*)
IF X > 20.0 THEN
	SIGMOID := 1.0;
ELSIF x < -85.0 THEN
	SIGMOID := 0.0;
ELSE
	SIGMOID := 1.0 / (1.0 + EXP(-X));
END_IF;


(* revision history
hm	10.12.2007		rev 1.0
	original version

hm	11. mar. 2008		rev 1.1
	extended range of valid inputs to +inv / -inv

hm 10. mar. 2009		rev 1.2
	real constants updated to new systax using dot																																																																																																																																																																																																																																																																																																																																																																																																																																																																																																																																																																																																																																																																																																																																																																																																																																																																																																																																																																																																																																																											

*)
END_FUNCTION

(* POU Mathematical/SIGN_I, ST *)
FUNCTION SIGN_I : BOOL
VAR_INPUT
	IN : DINT;
END_VAR


(*
version 1.3	27. oct. 2008
programmer 	hugo
tested by	tobias

this function return true if the integer input is negative

*)
SIGN_I := in.31;

(* revision history
hm 3.3.2007	rev 1.1
	changed method of function for better compatibility to other systems

hm	1.12.2007	rev 1.2
	changed code to improve performance

hm	27. oct. 2008	rev 1.3
	changed type of input to dint

*)
END_FUNCTION

(* POU Engineering/automation/SIGNAL, ST *)
FUNCTION_BLOCK SIGNAL
VAR_INPUT
	IN : BOOL;
	SIG : BYTE;
	TS : TIME;
END_VAR
VAR_OUTPUT
	Q : BOOL;
END_VAR
VAR
	tx: DWORD;
	step: BYTE;
END_VAR
VAR CONSTANT
	one : BYTE := 1;
END_VAR

(*
version 1.0	13 dec 2007
programmer 	hugo
tested by		tobias

this function generates an output signal according to a bit pattern SIG.
the patter is shifted to the output in time steps of TS.
ts defaults to 128 ms if not specified.
*)
IF in THEN
	(* an alarm is present read system time first *)
	tx := T_PLC_MS();
	(* calculate the step counter which is the lowest 3 bits of (time / ts) *)
	IF ts > t#0s THEN
		step := DWORD_TO_BYTE(tx / TIME_TO_DWORD(ts) AND 16#0000_0007);
	ELSE
		step := DWORD_TO_BYTE(SHR(tx,7) AND 16#0000_0007);
	END_IF;
	(* convert the value 0-7 in step into one bit only (bit 0-7) *)
	step := SHL(one,step);
	(* generate the output signal *)
	Q := (step AND sig) > 0;
ELSE
	Q := FALSE;
END_IF;

(* revision history
hm	13.12.2007		rev 1.0
	original version

*)
END_FUNCTION_BLOCK

(* POU Engineering/automation/SIGNAL_4, ST *)
FUNCTION_BLOCK SIGNAL_4
VAR_INPUT
	IN1 : BOOL;
	IN2 : BOOL;
	IN3 : BOOL;
	IN4 : BOOL;
	TS : TIME;
END_VAR
VAR_INPUT CONSTANT
	S1 : BYTE := 2#1111_1111;
	S2 : BYTE := 2#1111_0000;
	S3 : BYTE := 2#1010_1010;
	S4 : BYTE := 2#1010_0000;
END_VAR
VAR_OUTPUT
	Q : BOOL;
END_VAR
VAR
	sig : SIGNAL;
END_VAR

(*
version 1.0	13 dec 2007
programmer 	hugo
tested by		tobias

this function generates one out of 4 signals specified by bit patterns S1 .. S4.
the selected pattern will be shifted with the step time TS.
In1 has higher priority then In2 which has higher priority then IN3 and in4 has the lowest priority.
ts defaults to 128 ms if not specified.
*)
(* an alarm is present read system time first *)
(* check if an alarm is present if yes set sig to the alarm pattern otherwise exit the routine *)
IF in1 THEN
	sig(in := TRUE, sig := s1, TS := TS);
ELSIF in2 THEN
	sig(in := TRUE, sig := s2, TS := TS);
ELSIF in3 THEN
	sig(in := TRUE, sig := s3, TS := TS);
ELSIF in4 THEN
	sig(in := TRUE, sig := s4, TS := TS);
ELSE
	sig(in := FALSE);
END_IF;

(* set the output *)
Q := sig.Q;


(* revision history
hm	13.12.2007		rev 1.0
	original version

*)
END_FUNCTION_BLOCK

(* POU Mathematical/SINC, ST *)
FUNCTION SINC : REAL
VAR_INPUT
	X : REAL;
END_VAR


(*
version 1.2	10. mar. 2009
programmer 	hugo
tested by		tobias

this function calculates the sinc function.

*)
IF X = 0.0 THEN
	SINC := 1.0;
ELSE
	SINC := SIN(x) / x;
END_IF;


(* revision histroy
hm	11. mar. 2008	rev 1.0
	original version

hm	1.12.2007	rev 1.1
	changed code to improove performance

hm 10. mar. 2009	rev 1.2
	real constants updated to new systax using dot																																																																																																																																																																																																																																																																																																																																																																																																																																																																																																																																																																																																																																																																																																																																																																																																																																																																																																																																																																																																																																																											

*)
END_FUNCTION

(* POU Mathematical/Geometry/SPHERE_V, ST *)
FUNCTION SPHERE_V : REAL
VAR_INPUT
	rx : REAL;
END_VAR


(*
version 1.2	22. feb 2008
programmer 	hugo
tested by		tobias

sphere_V calculates the Volume of a Sphere


*)
sphere_V := 4.188790205 * Rx * RX * RX;

(* revision histroy
hm	16. oct 2007	rev 1.0
	original version

hm	4. dec 2007		rev 1.1
	changed code for better performance

hm	22. feb 2008		rev 1.2
	changed code for better performance
*)
END_FUNCTION

(* POU Logic/memory/STACK_16, ST *)
FUNCTION_BLOCK STACK_16
VAR_INPUT
	Din : DWORD;
	E : BOOL := TRUE;
	RD : BOOL;
	WD : BOOL;
	RST : BOOL;
END_VAR
VAR_OUTPUT
	Dout : DWORD;
	EMPTY : BOOL := TRUE;
	FULL : BOOL;
END_VAR
VAR
	stack : ARRAY[0..n] OF DWORD;
	pt : INT;
END_VAR
VAR CONSTANT
	n : INT := 15;	(* changing this value will chage the number of stored elements in the fifo *)
END_VAR


(*
version 2.0	25. jul 2009
programmer 	hugo
tested by		oscat

16 Dword STACK memory

*)
IF RST THEN
	(* asynchronous reset for the fifo *)
	pt := 0;
	EMPTY := TRUE;
	FULL := FALSE;
	Dout := 0;
ELSIF E THEN
	IF NOT EMPTY AND RD THEN
		(* read one element *)
		pt := pt - 1;
		Dout := stack[pt];
		EMPTY := pt = 0;
		FULL := FALSE;
	END_IF;
	IF NOT FULL AND WD THEN
		(* write one element *)
		stack[pt] := Din;
		pt := pt + 1;
		FULL := pt > n;
		EMPTY := FALSE;
	END_IF;
END_IF;


(* revision history
hm	4. aug. 2006	rev 1.0
	original version

hm	19. feb 2008	rev 1.1
	performance improvements

hm	17. oct. 2008	rev 1.2
	deleted unnecessary init with 0

hm	27. oct. 2008	rev 1.3
	optimized performance

hm	25. jul 2009	rev 2.0
	changed inputs to allow simultsaneous read and write
*)
END_FUNCTION_BLOCK

(* POU Logic/memory/STACK_32, ST *)
FUNCTION_BLOCK STACK_32
VAR_INPUT
	Din : DWORD;
	E : BOOL := TRUE;
	RD : BOOL;
	WD : BOOL;
	RST : BOOL;
END_VAR
VAR_OUTPUT
	Dout : DWORD;
	EMPTY : BOOL := TRUE;
	FULL : BOOL;
END_VAR
VAR
	stack : ARRAY[0..n] OF DWORD;
	pt : INT;
END_VAR
VAR CONSTANT
	n : INT := 31;	(* changing this value will chage the number of stored elements in the fifo *)
END_VAR


(*
version 2.0	25. jul 2009
programmer 	hugo
tested by		oscat

32 Dword STACK memory
*)
IF RST THEN
	(* asynchronous reset for the fifo *)
	pt := 0;
	EMPTY := TRUE;
	FULL := FALSE;
	Dout := 0;
ELSIF E THEN
	IF NOT EMPTY AND RD THEN
		(* read one element *)
		pt := pt - 1;
		Dout := stack[pt];
		EMPTY := pt = 0;
		FULL := FALSE;
	END_IF;
	IF NOT FULL AND WD THEN
		(* write one element *)
		stack[pt] := Din;
		pt := pt + 1;
		FULL := pt > n;
		EMPTY := FALSE;
	END_IF;
END_IF;


(* revision history
hm	4. aug. 2006	rev 1.0
	original version

hm	19. feb 2008	rev 1.1
	performance improvements

hm	17. oct. 2008	rev 1.2
	deleted unnecessary init with 0

ks	27. oct. 2008	rev 1.3
	optimized performance

hm	25. jul 2009	rev 2.0
	changed inputs to allow simultsaneous read and write

*)
END_FUNCTION_BLOCK

(* POU Engineering/signal processing/STAIR, ST *)
FUNCTION STAIR : REAL
VAR_INPUT
	X : REAL;
	D : REAL;
END_VAR


(*
version 1.4	10. mar. 2009
programmer 	oscat
tested by		tobias

the function stair converts an anlog input signal to a staircase like output.
D is the step width for the output signal.
if D = 0 then the output follows the input without a chage.
*) 
IF D > 0.0 THEN
	STAIR := DINT_TO_REAL(REAL_TO_DINT(X / D)) * D;
ELSE
	STAIR := X;
END_IF;



(* revision history
hm	28 jan 2007		rev 1.0
	original version

hm	27 dec 2007		rev 1.1
	changed code for better performance

hm	6. jan 2008		rev 1.2
	further performance improvement

hm	26. oct. 2008		rev 1.3
	optimized code

hm	10. mar. 2009	rev 1.4
	real constants updated to new systax using dot

*)
END_FUNCTION

(* POU Engineering/signal processing/STAIR2, ST *)
FUNCTION_BLOCK STAIR2
VAR_INPUT
	X : REAL;
	D : REAL;
END_VAR
VAR_OUTPUT
	Y: REAL;
END_VAR


(*
version 1.4	10. mar. 2009
programmer 	hugo
tested by		oscat

the function stair2 converts an anlog input signal to a staircase like output.
D is the step width for the output signal. the output will use D as a hysteresis for a stairchange.
if D = 0 then the output follows the input without a chage.
*) 
IF D > 0.0 THEN
	IF X >= Y + D OR X <= Y - D THEN Y := FLOOR(X/D) * D; END_IF;
ELSE
	Y := X;
END_IF;



(* revision history
hm	28 jan 2007		rev 1.0
	original version

hm	27. dec 2007	rev 1.1
	changed code for better performance

hm	30. jun. 2008	rev 1.2
	added type conversions to avoid warnings under codesys 3.0																																																																																																																																																																																																																																																											

ks	26. oct. 2008	rev 1.3
	improved code

hm	10. mar. 2009	rev 1.4
	real constants updated to new systax using dot

*)
END_FUNCTION_BLOCK

(* POU Logic/FF pulse triggered/STORE_8, ST *)
FUNCTION_BLOCK STORE_8
VAR_INPUT
	Set : BOOL;
	D0,D1, D2, D3, D4, D5, D6, D7 : BOOL;
	Clr : BOOL;
	Rst : BOOL;
END_VAR
VAR_OUTPUT
	Q0, Q1, Q2, Q3, Q4, Q5, Q6, Q7 : BOOL;
END_VAR
VAR
	edge: BOOL;
END_VAR

(*
version 1.2	14. mar. 2009
programmer 	hugo
tested by		oscat

Store_4 stores up to 4 boolean inputs until a reset is clearing the outputs.
the respective output is set with a true at the respective input and stays true until a reset is generated.
a set input is used to set all outputs true at the same time, independent of their inputs.
a clear input is used to reset only the lowest priority of the outputs one at a time.
the lowest priority is q3.

*)
IF rst OR set THEN
	q0 := NOT rst;
	q1 := q0;
	q2 := q0;
	q3 := q0;
	q4 := q0;
	q5 := q0;
	q6 := q0;
	q7 := q0;
ELSE
	IF D0 THEN Q0 := TRUE; END_IF;
	IF D1 THEN Q1 := TRUE; END_IF;
	IF D2 THEN Q2 := TRUE; END_IF;
	IF D3 THEN Q3 := TRUE; END_IF;
	IF D4 THEN Q4 := TRUE; END_IF;
	IF D5 THEN Q5 := TRUE; END_IF;
	IF D6 THEN Q6 := TRUE; END_IF;
	IF D7 THEN Q7 := TRUE; END_IF;

	IF clr AND NOT edge THEN
		IF q0 THEN q0 := FALSE;
		ELSIF q1 THEN q1 := FALSE;
		ELSIF q2 THEN q2 := FALSE;
		ELSIF q3 THEN q3 := FALSE;
		ELSIF q4 THEN q4 := FALSE;
		ELSIF q5 THEN q5 := FALSE;
		ELSIF q6 THEN q6 := FALSE;
		ELSE q7 := FALSE;
		END_IF;
	END_IF;
	edge := clr;
END_IF;


(* revision history
hm	25.12.2007	rev 1.0
	original version

hm	30. oct. 2008	rev 1.1
	optimized performance

hm	14. mar. 2009	rev 1.2
	removed double assignments

*)
END_FUNCTION_BLOCK

(* POU Logic/gate logic/SWAP_BYTE, ST *)
FUNCTION SWAP_BYTE : WORD
VAR_INPUT
	IN : WORD;
END_VAR


(*
version 1.0	4 feb 2008
programmer 	hugo
tested by		tobias

This function swaps the high and low byte of the word in.

*)
SWAP_BYTE := ROL(in,8);


(* revision history
hm		4. feb 2008	rev 1.0
	original version

*)
END_FUNCTION

(* POU Logic/gate logic/SWAP_BYTE2, ST *)
FUNCTION SWAP_BYTE2 : DWORD
VAR_INPUT
	IN : DWORD;
END_VAR


(*
version 1.0	4 feb 2008
programmer 	hugo
tested by		tobias

This function reverses the byte order in the dword.

*)
Swap_Byte2 := (ROR(in,8) AND 16#FF00FF00) OR (ROL(in,8) AND 16#00FF00FF);

(* revision history
hm		4. feb 2008	rev 1.0
	original version

*)
END_FUNCTION

(* POU Mathematical/TANC, ST *)
FUNCTION TANC : REAL
VAR_INPUT
	X : REAL;
END_VAR


(*
version 1.1	10. mar. 2009
programmer 	hugo
tested by		oscat

this function calculates the tanc function.

*)
IF X = 0.0 THEN
	TANC := 1.0;
ELSE
	TANC := TAN(x) / x;
END_IF;


(* revision histroy
hm	23. oct. 2008	rev 1.0
	original version

hm 10. mar. 2009	rev 1.1
	real constants updated to new systax using dot																																																																																																																																																																																																																																																																																																																																																																																																																																																																																																																																																																																																																																																																																																																																																																																																																																																																																																																																																																																																																																																											

*)
END_FUNCTION

(* POU Mathematical/TANH, ST *)
FUNCTION TANH : REAL
VAR_INPUT
	X : REAL;
END_VAR


(*
version 1.3	10. mar. 2009
programmer 	hugo
tested by		tobias

this function calculates the tangens hyperbolicus

*)
IF X > 20.0 THEN
	TANH := 1.0;
ELSIF X < -20.0 THEN
	TANH := -1.0;
ELSE
	TANH := 1.0 - 2.0 / (EXP(2.0 * x) + 1.0);
END_IF;


(* revision hisdtory
hm		12.1.2007		rev 1.0
	original version

hm		1.12.2007		rev 1.1
	changed code to improve performance

hm		10. mar 2008	rev 1.2
	corrected an error in formula
	extended range of valid inputs to +/- INV

hm 10. mar. 2009	rev 1.3
	real constants updated to new systax using dot																																																																																																																																																																																																																																																																																																																																																																																																																																																																																																																																																																																																																																																																																																																																																																																																																																																																																																																																																																																																																																																											

*)
END_FUNCTION

(* POU Engineering/measurements/TC_MS, ST *)
FUNCTION_BLOCK TC_MS

VAR_OUTPUT
	TC : DWORD;
END_VAR
VAR
	init: BOOL;
	tx: DWORD;
	last: DWORD;
END_VAR

(*
	version 1.0	13 mar 2008
	programmer 	hugo
	tested by		tobias

TC_MS delivers the time it was last called on the output TC in Milliseconds.

*)
(* read system timer *)
tx := T_PLC_MS();

IF NOT init THEN
	init := TRUE;
	TC := 0;
ELSE
	tc := tx - last;
END_IF;
last := tx;

(* revision history
hm		13. mar. 2008	rev 1.0
	original version

*)
END_FUNCTION_BLOCK

(* POU Engineering/measurements/TC_US, ST *)
FUNCTION_BLOCK TC_US

VAR_OUTPUT
	TC : DWORD;
END_VAR
VAR
	init: BOOL;
	tx: DWORD;
	last: DWORD;
END_VAR

(*
	version 1.0	13 mar 2008
	programmer 	hugo
	tested by		tobias

TC_US delivers the time it was last called on the output TC in Microseconds.

*)
(* read system timer *)
tx := T_PLC_US();

IF NOT init THEN
	init := TRUE;
	TC := 0;
ELSE
	tc := tx - last;
END_IF;
last := tx;

(* revision history
hm		13. mar. 2008	rev 1.0
	original version

*)
END_FUNCTION_BLOCK

(* POU Engineering/sensor/TEMP_NI, ST *)
FUNCTION TEMP_NI : REAL
VAR_INPUT
	Res : REAL;
	R0 : REAL;
END_VAR


(*
version 1.5	10. mar. 2009
programmer 	hugo
tested by		tobias

this function returns the temperature for a nickel sensor in a range from -60..+180 °C *)
TEMP_NI := (SQRT(0.30085225 - 2.66E-3 * (R0 - Res)) - 0.5485) * 751.8796992;


(* revision history

hm 24.1.2007		rev 1.1
	deleted unused variable A, B, C

hm 10.9.2007		rev 1.2
	changed accuracy to 0.02 degrees to improove performace

hm 17. 12 2007	rev 1.3
	improovements for better performance and higher accuracy

hm	6. jan 2008	rev 1.4
	further performance improvement

hm	10. mar. 2009	rev 1.5
	removed nested comments

*)
END_FUNCTION

(* POU Engineering/sensor/TEMP_NTC, ST *)
FUNCTION TEMP_NTC : REAL
VAR_INPUT
	RES : REAL;
	RN : REAL;
	B : REAL;
END_VAR


(*
version 1.1	11. mar. 2009
programmer 	hugo
tested by		tobias

this function returs the temperature for a NTC sensor for a range from 0..85 °C.
RN is the resistance at 25 °C and B is a constant for the given sensor.

*)
IF res > 0.0 THEN
	TEMP_NTC := B * 298.15 / (B + LN(RES / RN) * 298.15) -273.15;
END_IF;


(* revision history

hm 30. dec. 2008	rev 1.0
	original version

hm	11. mar. 2009	rev 1.1
	changed real constants to use dot syntax

*)
END_FUNCTION

(* POU Engineering/sensor/TEMP_PT, ST *)
FUNCTION TEMP_PT : REAL
VAR_INPUT
	Res : REAL;
	R0 : REAL;
END_VAR
VAR CONSTANT
	A : REAL := 3.9083E-3 ;
	B : REAL := -5.775E-7;
	accuracy : REAL := 0.01;
END_VAR
VAR
	step: REAL := 50.0;
	X: REAL;
	Y: REAL;
	t1: REAL;
	pt : POINTER TO DWORD;
END_VAR

(*
version 1.7	11. mar. 2009
programmer 	hugo
tested by		oscat

this function returs the temperature for a platinum sensor for a range from -200..+850 °C *)
X := A * R0;
Y := B * R0;
IF Res >= R0 THEN
	t1 := X * X - 4.0 * Y * (R0 - Res);
	IF t1 < 0.0 THEN
		TEMP_PT := 10000.0;
	ELSE
		TEMP_PT := (-X + SQRT(t1)) / (2.0 * Y);
	END_IF;
ELSE
	pt := ADR(step);
	(* since the formula cannot be solved this is a successive approximation *)
	TEMP_PT := -100.0;
	WHILE step > accuracy DO
		(* test if result greater or less *)
		IF RES_PT(TEMP_PT, R0) < res THEN TEMP_PT := TEMP_PT + step; ELSE TEMP_PT := TEMP_PT - step; END_IF;
		pt^ := pt^ - 8388608;  (* this is a super fast divide by 2 method for non floating point CPUs *)
		(* the alternative code: step := step * 0.5; *)
	END_WHILE;
END_IF;

(* revision history

rev 1.1 hm 24.1.2007	
	deleted unused variable C

rev 1.2 hm 10.9.2007
	reduced accuracy to 0.02 to shorten execution time

rev 1.3	hm	2. dec 2007
	changed code for better performance

rev	1.4	hm	23. dec 2007
	avoid a negative square root if input values are wrong

rev 1.5 hm	5. jan 2008
	replaced / 2 with * 0.5 for better performance

hm	31. oct. 2008	rev 1.6
	improved performance

hm	11. mar. 2009	rev 1.7
	changed real constants to use dot syntax

*)
END_FUNCTION

(* POU Engineering/sensor/TEMP_SI, ST *)
FUNCTION TEMP_SI : REAL
VAR_INPUT
	Res : REAL;
	RS : REAL;
	TS : REAL;
END_VAR


(*
version 1.5	10. mar. 2009
programmer 	hugo
tested by		tobias

this function returs the temperature for a silicon sensor for a range from -60..+180 °C
for example KTY10 RS at TS normally 25 °C
*)
TEMP_SI := (-7.64E-3 + SQRT(Res / RS * 6.64E-5 - 0.803E-5)) * 30120.48193 + TS;



(* revision history

hm 24.1.2007		rev 1.1
	the function would only work for TS = 25, now it works for other values of ts.

hm 10.9.2007		rev 1.2
	changed the function to use successive approcimation to avoid an error generated by a sqrt from a negative result.
	changed accuracy to 0.02 degrees to shorten execution time

hm 17. 12 2007	rev 1.3
	improovements for better performance

hm	6. jan 2008	rev 1.4
	further performance improvement

hm	10. mar. 2009	rev 1.5
	removed nested comments

*)
END_FUNCTION

(* POU Engineering/conversion/TEMPERATURE, ST *)
FUNCTION_BLOCK TEMPERATURE
VAR_INPUT
	K : REAL;
	C : REAL := -273.15;
	F : REAL := -459.67;
	Re : REAL := -218.52;
	Ra : REAL;
END_VAR
VAR_OUTPUT
	YK : REAL;
	YC : REAL;
	YF : REAL;
	YRe : REAL;
	YRa : REAL;
END_VAR


(*
version 1.0	21 feb 2008
programmer 	hugo
tested by	oscat

this function converts different temperature units
any unused input can simply be left open.
different inputs connected at the same time will be added up.

*)
YK := K + (C + 273.15) + (F + 459.67) * 0.555555555555 + (Re * 1.25 + 273.15) + (Ra * 0.555555555555);
YC := YK -273.15;
YF := YK * 1.8 - 459.67;
YRe := (YK - 273.15) * 0.8;
YRa := YK * 1.8;


(* revision history
hm	21. feb. 2008	rev 1.0
	original version

*)
END_FUNCTION_BLOCK

(* POU X_TEST/TEST_ARRAY_SORT, ST *)
FUNCTION_BLOCK TEST_ARRAY_SORT
VAR_INPUT
END_VAR
VAR_OUTPUT
END_VAR
VAR CONSTANT
	array_max : INT := 999;
END_VAR
VAR
	buffer : ARRAY[0..array_max] OF REAL;
	i: INT;
	tx: TIME;
	t_sort : TIME;
END_VAR
(* prefill array *)
buffer[0] := 0.0;
buffer[1] := 1.0;
buffer[2] := 0.0;
buffer[3] := -100.0;
buffer[4] := 100.0;

FOR i := 5 TO ARRAY_MAX DO
	buffer[i] := INT_TO_REAL(i)-20.0;
END_FOR;

_ARRAY_SHUFFLE(ADR(buffer), SIZEOF(buffer));
tx := TIME();
_ARRAY_SORT(ADR(buffer), SIZEOF(buffer));
t_sort := TIME() - tx;
END_FUNCTION_BLOCK

(* POU X_TEST/TEST_CRC_GEN, ST *)
FUNCTION_BLOCK TEST_CRC_GEN
VAR_INPUT
END_VAR
VAR_OUTPUT
	ERROR : BOOL;
	info : STRING (10);
END_VAR
VAR
	BUFFER : ARRAY[0..8] OF BYTE := 16#31, 16#32, 16#33, 16#34, 16#35, 16#36, 16#37, 16#38, 16#39;
	pt : POINTER TO ARRAY[0..100] OF BYTE;
	size : INT;
	erg: DWORD;
END_VAR
pt := ADR(buffer);
size := SIZEOF(buffer);

erg := CRC_GEN(pt, size, 3, 16#3, 16#7, TRUE, TRUE, 16#0);
IF erg <> 16#6 THEN
	error := TRUE;
	info := 'CRC-3/ROHC';
END_IF;

erg := CRC_GEN(pt, size, 5, 16#9, 16#9, FALSE, FALSE, 16#0);
IF erg <> 16#0 THEN
	error := TRUE;
	info := 'CRC-5/EPC';
END_IF;

erg := CRC_GEN(pt, size, 6, 16#19, 16#0, TRUE, FALSE, 16#0);
IF erg <> 16#19 THEN
	error := TRUE;
	info := 'CRC-6/DARC';
END_IF;

erg := CRC_GEN(pt, size, 7, 16#4F, 16#7F, TRUE, TRUE, 16#0);
IF erg <> 16#53 THEN
	error := TRUE;
	info := 'CRC-7/ROHC';
END_IF;

erg := CRC_GEN(pt, size, 8, 16#1D, 16#FD, FALSE, FALSE, 16#0);
IF erg <> 16#7E THEN
	error := TRUE;
	info := 'CRC-8/I-CODE';
END_IF;

erg := CRC_GEN(pt, size, 10, 16#233, 16#000, FALSE, FALSE, 16#0);
IF erg <> 16#199 THEN
	error := TRUE;
	info := 'CRC-10';
END_IF;

erg := CRC_GEN(pt, size, 12, 16#80F, 16#000, FALSE, TRUE, 16#0);
IF erg <> 16#DAF THEN
	error := TRUE;
	info := 'CRC-12/3GPP';
END_IF;

erg := CRC_GEN(pt, size, 14, 16#0805, 16#000, TRUE, TRUE, 16#0);
IF erg <> 16#082D  THEN
	error := TRUE;
	info := 'CRC-14/DARC';
END_IF;

erg := CRC_GEN(pt, size, 15, 16#4599, 16#000, FALSE, FALSE, 16#0);
IF erg <> 16#059E  THEN
	error := TRUE;
	info := 'CRC-15';
END_IF;

erg := CRC_GEN(pt, size, 16, 16#8BB7, 16#000, FALSE, FALSE, 16#0);
IF erg <> 16#D0DB  THEN
	error := TRUE;
	info := 'CRC-16/T10-DIF';
END_IF;

erg := CRC_GEN(pt, size, 24, 16#5D6DCB, 16#ABCDEF, FALSE, FALSE, 16#0);
IF erg <> 16#1F23B8  THEN
	error := TRUE;
	info := 'CRC-24/FLEXRAY-B';
END_IF;

erg := CRC_GEN(pt, size, 32, 16#04C11DB7, 16#FFFFFFFF, TRUE, TRUE, 16#0);
IF erg <> 16#340BC6D9  THEN
	error := TRUE;
	info := 'JAMCRC';
END_IF;



(*
   Name   : "CRC-82/DARC"
   Width  : 82
   Poly   : 0308C0111011401440411
   Init   : 000000000000000000000
   RefIn  : True
   RefOut : True
   XorOut : 000000000000000000000
   Check  : 09EA83F625023801FD612
	pt : POINTER TO ARRAY[1..32000] OF BYTE;
	size : UINT;
	Polynom_L : DWORD;
	Polynom_32 : BOOL;
	init: DWORD;
	XOR_out : DWORD;
	rev_in : BOOL;
	rev_out : BOOL;

*)
END_FUNCTION_BLOCK

(* POU X_TEST/test_date, ST *)
FUNCTION_BLOCK test_date
VAR_INPUT
END_VAR
VAR_OUTPUT
	error: BOOL;
END_VAR
VAR
	test : DWORD;
	c_date : DATE;
	x_date : DATE;
	c_day : INT;
	c_month : INT;
	c_year : INT;
	d_str : STRING;
END_VAR
c_date := DWORD_TO_DATE(test);
d_str := DATE_TO_STRING(c_date);
c_year := STRING_TO_INT(MID(d_str, 4, 3));
c_month := STRING_TO_INT(MID(d_str, 2, 8));
c_day := STRING_TO_INT(MID(d_str, 2, 11));


(* test leap_day *)
IF LEAP_DAY(c_date)  XOR (c_day = 29 AND c_month = 2) THEN error := TRUE; END_IF;

(* test set_date *)
x_date := SET_DATE(c_year, c_month, c_day);
IF x_date <> c_date THEN error := TRUE; END_IF;

(* test year_end *)
IF SET_DATE(c_year, 12, 31) <> YEAR_END(c_year) THEN error := TRUE; END_IF;

(* test year begin  and day_of_year *)
x_date := YEAR_BEGIN(c_year);
IF SET_DATE(c_year, 1, 1) <> x_date THEN error := TRUE; END_IF;
(* test day_of_year *)
IF UDINT_TO_DATE(DATE_TO_UDINT(x_date) + (DAY_OF_YEAR(c_date) - 1) * 86400) <> c_date THEN error := TRUE; END_IF;

(* test leap_year *)
IF LEAP_OF_DATE(c_DATE) <> (SHL(c_year,14) = 0) THEN error := TRUE; END_IF;



(* next test to date *)
IF NOT error THEN
	IF test < DATE_TO_DWORD(D#2099-12-31) THEN test := test + 86400; END_IF;
END_IF;
END_FUNCTION_BLOCK

(* POU Time&Date/YEAR_END, ST *)
FUNCTION YEAR_END : DATE
VAR_INPUT
	y : INT;
END_VAR


(*
version 1.1	24. jan. 2011
programmer 	hugo
tested by	oscat

returs the date of december 31st for the given year  
the function works for dates from 1970 - 2099 

*)
YEAR_END := DWORD_TO_DATE(SHR(INT_TO_DWORD(y) * 1461 - 2876712, 2) * 86400);



(* revision history
hm	15. jun. 2008	rev 1.0
	original version

hm	24. jan 2011	rev 1.1
	improved performance
*)
END_FUNCTION

(* POU X_TEST/test_date_add, ST *)
FUNCTION_BLOCK test_date_add
VAR_INPUT
END_VAR
VAR_OUTPUT
	error: BOOL;
END_VAR
VAR
END_VAR
IF DATE_ADD(D#2011-03-22,-1,0,0,0) <> D#2011-3-21 THEN error := TRUE; END_IF;
IF DATE_ADD(D#2011-03-22,0,0,0,0) <> D#2011-3-22 THEN error := TRUE; END_IF;
IF DATE_ADD(D#2011-03-22,-1,-1,-1,-1) <> D#2010-2-14 THEN error := TRUE; END_IF;
IF DATE_ADD(D#2011-03-22,1,1,1,1) <> D#2012-4-30 THEN error := TRUE; END_IF;
IF DATE_ADD(D#2011-03-22,366,0,0,0) <> D#2012-3-22 THEN error := TRUE; END_IF;
IF DATE_ADD(D#2011-03-22,0,0,13,0) <> D#2012-4-22 THEN error := TRUE; END_IF;
IF DATE_ADD(D#2011-03-22,0,0,-13,0) <> D#2010-2-22 THEN error := TRUE; END_IF;
END_FUNCTION_BLOCK

(* POU X_TEST/test_fact, ST *)
FUNCTION_BLOCK test_fact
VAR_INPUT
END_VAR
VAR_OUTPUT
END_VAR
VAR
	fx : ARRAY[0..12] OF DINT := 1,1,2,6,24,120,720,5040,40320,362880,3628800,39916800,479001600;
	tmp, tx: TIME;
	i: INT;
	j: INT;
END_VAR
VAR_OUTPUT
	error: BOOL;
	ty : TIME := t#1h;
END_VAR
tmp := TIME();
IF error THEN RETURN; END_IF;
FOR j := 1 TO 100 DO
	FOR i := 0 TO 12 DO
		IF fx[i] <> FACT(i) THEN error := TRUE; END_IF;
	END_FOR;
END_FOR;
tx := TIME() - tmp;
ty := MIN(tx, ty);
END_FUNCTION_BLOCK

(* POU X_TEST/test_filter_w, CFC *)
FUNCTION_BLOCK test_filter_w
VAR_INPUT
END_VAR
VAR_OUTPUT
END_VAR
VAR
	aa: FILTER_W;
END_VAR
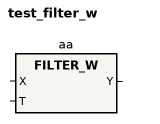
_CFC_ (* Continuous Function Chart, elements in execution order *)
#0 aa:FILTER_W(X: -, T: -)
_END_CFC_
(* the same logic as Structured Text *)
aa();
END_FUNCTION_BLOCK

(* POU X_TEST/test_flow_meter, CFC *)
FUNCTION_BLOCK test_flow_meter
VAR_INPUT
END_VAR
VAR_OUTPUT
END_VAR
VAR
	x: REAL;
	y: UDINT;
	xx: FLOW_METER;
	xy: TP;
	EX: BOOL;
	et: TIME := T#10s;
	EP: BOOL;
	VX: REAL := 400;
	RST: BOOL;
	F: REAL;
END_VAR
VAR (* helpers for the ST form of the networks *)
	_t8 : BOOL;
END_VAR
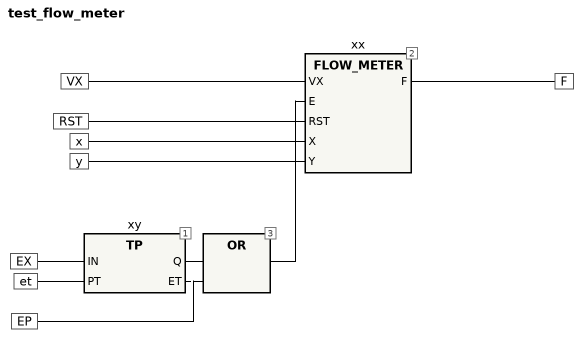
_CFC_ (* Continuous Function Chart, elements in execution order *)
#0 F <= #2.F
#1 xy:TP(IN: EX, PT: et)
#2 xx:FLOW_METER(VX: VX, E: #3, RST: RST, X: x, Y: y)
#3 OR(#1.Q, EP)
_END_CFC_
(* the same logic as Structured Text *)
F := xx.F;
xy(IN := EX, PT := et);
xx(VX := VX, E := _t8, RST := RST, X := x, Y := y);
_t8 := xy.Q OR EP;
END_FUNCTION_BLOCK

(* POU X_TEST/TEST_GCD, ST *)
FUNCTION_BLOCK TEST_GCD
VAR_INPUT
END_VAR
VAR_OUTPUT
	error : BOOL;
END_VAR
VAR
END_VAR
IF GCD(12,18) <> 6 THEN error := TRUE; END_IF;
IF GCD(0,18) <> 18 THEN error := TRUE; END_IF;
IF GCD(12,0) <> 12 THEN error := TRUE; END_IF;
IF GCD(0,0) <> 0 THEN error := TRUE; END_IF;
IF GCD(12,132) <> 12 THEN error := TRUE; END_IF;
IF GCD(12,36) <> 12 THEN error := TRUE; END_IF;
IF GCD(12,90) <> 6 THEN error := TRUE; END_IF;
IF GCD(1,1) <> 1 THEN error := TRUE; END_IF;
IF GCD(2,1) <> 1 THEN error := TRUE; END_IF;
IF GCD(2,7) <> 1 THEN error := TRUE; END_IF;
IF GCD(2,18) <> 2 THEN error := TRUE; END_IF;
IF GCD(3,18) <> 3 THEN error := TRUE; END_IF;
IF GCD(3,7) <> 1 THEN error := TRUE; END_IF;
IF GCD(3528,3780) <> 252 THEN error := TRUE; END_IF;
IF GCD(1071,1029) <> 21 THEN error := TRUE; END_IF;
IF GCD(-12,132) <> 12 THEN error := TRUE; END_IF;
IF GCD(12,-36) <> 12 THEN error := TRUE; END_IF;
END_FUNCTION_BLOCK

(* POU X_TEST/TEST_HOLIDAY, CFC *)
FUNCTION_BLOCK TEST_HOLIDAY
VAR_INPUT
END_VAR
VAR_OUTPUT
END_VAR
VAR
	cc: HOLIDAY;
	t_date: DATE := D#2011-04-22;
	langw: INT := 4;
	friday: BOOL;
	saturday: BOOL;
	sunday: BOOL;
	holi: BOOL;
	name: STRING(30);
	HOLIDAY_DE : ARRAY[0..29] OF HOLIDAY_DATA := (name := 'Neujahr', day := 1, month := 1, use := 1),
		(name := 'Heilig Drei Könige', day := 6, month := 1, use := 1),
		(name := 'Karfreitag', day := -2, month := 0, use := 1),
		(name := 'Ostersonntag', day := 0, month := 0, use := 1),
		(name := 'Ostermontag', day := 1, month := 0, use := 1),
		(name := 'Tag der Arbeit', day := 1, month := 5, use := 1),
		(name := 'Christi Himmelfahrt', day := 39, month := 0, use := 1),
		(name := 'Pfingstsonntag', day := 49, month := 0, use := 1),
		(name := 'Pfingstmontag', day := 50, month := 0, use := 1),
		(name := 'Fronleichnam', day := 60, month := 0, use := 1),
		(name := 'Augsburger Friedensfest', day := 8, month := 8, use := 0),
		(name := 'Maria Himmelfahrt', day := 15, month := 8, use := 1),
		(name := 'Tag der Deutschen Einheit', day := 3, month := 10, use := 1),
		(name := 'Reformationstag', day := 31, month := 10, use := 0),
		(name := 'Allerheiligen', day := 1, month := 11, use := 1),
		(name := 'Buss und Bettag', day := 23, month := 11, use := 0),
		(name := '1. Weihnachtstag', day := 25, month := 12, use := 1),
		(name := '2. Weihnachtstag', day := 26, month := 12, use := 1);


	(*	if month = 0 then F_day is the offset in days from easter
		used :0 = NOT used, 1 = used, -1..-7 menas the weekday before the specified DATE example -3 means wednesday before 23.11
	*)

	HOLIDAY_AT : ARRAY[0..29] OF HOLIDAY_DATA := (name := 'Neujahr', day := 1, month := 1, use := 1),
		(name := 'Heilig Drei Könige', day := 6, month := 1, use := 1),
		(name := 'Karfreitag', day := -2, month := 0, use := 1),
		(name := 'Ostersonntag', day := 0, month := 0, use := 1),
		(name := 'Ostermontag', day := 1, month := 0, use := 1),
		(name := '', day := 1, month := 5, use := 0),
		(name := 'Christi Himmelfahrt', day := 39, month := 0, use := 1),
		(name := 'Pfingstsonntag', day := 49, month := 0, use := 1),
		(name := 'Pfingstmontag', day := 50, month := 0, use := 1),
		(name := 'Fronleichnam', day := 60, month := 0, use := 1),
		(name := '', day := 8, month := 8, use := 0),
		(name := 'Maria Himmelfahrt', day := 15, month := 8, use := 1),
		(name := '', day := 3, month := 10, use := 0),
		(name := '', day := 31, month := 10, use := 0),
		(name := 'Allerheiligen', day := 1, month := 11, use := 1),
		(name := 'Maria Empfängnis', day := 8, month := 12, use := 1),
		(name := '1. Weihnachtstag', day := 25, month := 12, use := 1),
		(name := '2. Weihnachtstag', day := 26, month := 12, use := 1);

	HOLIDAY_FR : ARRAY[0..29] OF HOLIDAY_DATA := (name := 'Nouvel an', day := 1, month := 1, use := 1),
		(name := 'St Valentin', day := 14, month := 2, use := 0),
		(name := 'Vendredi Saint (alsace)', day := -2, month := 0, use := 0),
		(name := 'Dimanche de pâques', day := 0, month := 0, use := 1),
		(name := 'Lundi de pâques', day := 1, month := 0, use := 1),
		(name := 'Jeudi de Ascension', day := 39, month := 0, use := 1),
		(name := 'dimanche de Pentecôte ', day := 49, month := 0, use := 1),
		(name := 'jeudi de la Trinité', day := 60, month := 0, use := 0),
		(name := 'Fête du travail', day := 1, month := 5, use := 1),
		(name := 'Victoire 1945 ', day := 8, month := 5, use := 1),
		(name := 'Prise de La bastille', day := 14, month := 7, use := 1),
		(name := '15 Août 1944', day := 15, month := 8, use := 1),
		(name := 'Halloween', day := 31, month := 10, use := 0),
		(name := 'Armistice 1918', day := 11, month := 11, use := 1),
		(name := 'Noël', day := 25, month := 12, use := 1),
		(name := 'Saint Étienne (alsace)', day := 26, month := 12, use := 0),
		(name := 'Fête de la musique', day := 21, month := 6, use := 0);


	HOLIDAY_BED : ARRAY[0..29] OF HOLIDAY_DATA :=	(name := 'Neujahr', day := 1, month := 1, use := 1),
		(name := 'Ostersonntag', day := 0, month := 0, use := 1),
		(name := 'Ostermontag', day := 1, month := 0, use := 1),
		(name := 'Tag der Arbeit', day := 1, month := 5, use := 1),
		(name := 'Christi Himmelfahrt', day := 39, month := 0, use := 1),
		(name := 'Pfingsten', day := 49, month := 0, use := 1),
		(name := 'Pfingstmontag', day := 50, month := 0, use := 1),
		(name := 'Nationalfeiertag', day := 21, month := 7, use := 1),
		(name := 'Mariä Himmelfahrt', day := 15, month := 8, use := 1),
		(name := 'Allerheiligen', day := 1, month := 11, use := 1),
		(name := 'Feiertag DG', day := 15, month := 11, use := 1),
		(name := 'Heiligabend', day := 24, month := 12, use := 1),
		(name := '1. Weihnachtstag', day := 25, month := 12, use := 1),
		(name := '2. Weihnachtstag', day := 26, month := 12, use := 1),
		(name := 'Silvester', day := 31, month := 12, use := 1);


	HOLIDAY_ITD : ARRAY[0..29] OF HOLIDAY_DATA := (name := 'Neujahr', day := 1, month := 1, use := 1),
		(name := 'Heilig Drei Könige', day := 6, month := 1, use := 1),
		(name := 'Ostersonntag', day := 0, month := 0, use := 1),
		(name := 'Ostermontag', day := 1, month := 0, use := 1),
		(name := 'Tag der Befeiung Italiens', day := 25, month := 4, use := 1),
		(name := 'Tag der Arbeit', day := 1, month := 5, use := 1),
		(name := 'Pfingsten', day := 49, month := 0, use := 1),
		(name := 'Pfingstmontag', day := 50, month := 0, use := 1),
		(name := 'Tag der Republik Italien', day := 2, month := 6, use := 1),
		(name := 'Mariä Himmelfahrt', day := 15, month := 8, use := 1),
		(name := 'Allerheiligen', day := 1, month := 11, use := 1),
		(name := 'Mariä Empfängnis', day := 8, month := 12, use := 1),
		(name := 'Heiligabend', day := 24, month := 12, use := 0),
		(name := '1. Weihnachtstag', day := 25, month := 12, use := 1),
		(name := '2. Stephanstag', day := 26, month := 12, use := 1);


END_VAR
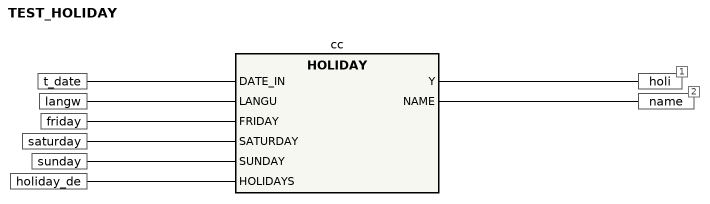
_CFC_ (* Continuous Function Chart, elements in execution order *)
#0 cc:HOLIDAY(DATE_IN: t_date, LANGU: langw, FRIDAY: friday, SATURDAY: saturday, SUNDAY: sunday, HOLIDAYS: holiday_de)
#1 holi <= #0.Y
#2 name <= #0.NAME
_END_CFC_
(* the same logic as Structured Text *)
cc(DATE_IN := t_date, LANGU := langw, FRIDAY := friday, SATURDAY := saturday, SUNDAY := sunday, HOLIDAYS := holiday_de);
holi := cc.Y;
name := cc.NAME;
END_FUNCTION_BLOCK

(* POU X_TEST/test_list_clean_add_get_len, ST *)
FUNCTION_BLOCK test_list_clean_add_get_len
VAR_INPUT
END_VAR
VAR_OUTPUT
	error : BOOL;
END_VAR
VAR
	L1 : STRING(LIST_LENGTH);
	tmp: BYTE;
END_VAR
IF error THEN RETURN; END_IF;
L1 := '';
tmp := CODE('§',1);
IF LIST_LEN(tmp,L1) <> 0 THEN error := TRUE; END_IF;
LIST_ADD(tmp,'',L1);	(* add one empty element *)
IF LIST_LEN(tmp,L1) <> 1 THEN error := TRUE; END_IF;
LIST_ADD(tmp,'a',L1);	(* add one empty element *)
IF LIST_LEN(tmp,L1) <> 2 THEN error := TRUE; END_IF;
LIST_ADD(tmp,'bbb',L1);	(* add one empty element *)
IF LIST_LEN(tmp,L1) <> 3 THEN error := TRUE; END_IF;
LIST_ADD(tmp,'',L1);	(* add one empty element *)
IF LIST_LEN(tmp,L1) <> 4 THEN error := TRUE; END_IF;
LIST_ADD(tmp,'',L1);	(* add one empty element *)
IF LIST_LEN(tmp,L1) <> 5 THEN error := TRUE; END_IF;
LIST_ADD(tmp,'cc',L1);	(* add one empty element *)
IF LIST_LEN(tmp,L1) <> 6 THEN error := TRUE; END_IF;
LIST_ADD(tmp,'',L1);	(* add one empty element *)
IF LIST_LEN(tmp,L1) <> 7 THEN error := TRUE; END_IF;
IF L1 <> '§§a§bbb§§§cc§' THEN error := TRUE; END_IF;
IF LIST_GET(tmp,0,L1) <> '' THEN error := TRUE; END_IF;
IF LIST_GET(tmp,1,L1) <> '' THEN error := TRUE; END_IF;
IF LIST_GET(tmp,2,L1) <> 'a' THEN error := TRUE; END_IF;
IF LIST_GET(tmp,3,L1) <> 'bbb' THEN error := TRUE; END_IF;
IF LIST_GET(tmp,4,L1) <> '' THEN error := TRUE; END_IF;
IF LIST_GET(tmp,5,L1) <> '' THEN error := TRUE; END_IF;
IF LIST_GET(tmp,6,L1) <> 'cc' THEN error := TRUE; END_IF;
IF LIST_GET(tmp,7,L1) <> '' THEN error := TRUE; END_IF;
IF LIST_GET(tmp,8,L1) <> '' THEN error := TRUE; END_IF;
LIST_CLEAN(tmp,L1);
IF L1 <> '§a§bbb§cc' THEN error := TRUE; END_IF;
L1 := '';
LIST_CLEAN(tmp,L1);
IF L1 <> '' THEN error := TRUE; END_IF;
L1 := '§';
LIST_CLEAN(tmp,L1);
IF L1 <> '' THEN error := TRUE; END_IF;
END_FUNCTION_BLOCK

(* POU X_TEST/test_list_insert, ST *)
FUNCTION_BLOCK test_list_insert
VAR_INPUT
END_VAR
VAR_OUTPUT
	error : BOOL;
END_VAR
VAR
	L1 : STRING(LIST_LENGTH);
	tmp: BYTE;
END_VAR
IF error THEN RETURN; END_IF;
L1 := '';
tmp := CODE('§',1);
LIST_INSERT(tmp, 1, '', L1);
IF L1 <> '§' THEN error := TRUE; END_IF;
L1 := '';
LIST_INSERT(tmp, 1, 'a', L1);
IF L1 <> '§a' THEN error := TRUE; END_IF;
LIST_INSERT(tmp, 1, '', L1);
IF L1 <> '§§a' THEN error := TRUE; END_IF;
LIST_INSERT(tmp, 1, 'b', L1);
IF L1 <> '§b§§a' THEN error := TRUE; END_IF;
LIST_INSERT(tmp, 2, 'c', L1);
IF L1 <> '§b§c§§a' THEN error := TRUE; END_IF;
LIST_INSERT(tmp, 4, 'd', L1);
IF L1 <> '§b§c§§d§a' THEN error := TRUE; END_IF;
LIST_INSERT(tmp, 6, 'e', L1);
IF L1 <> '§b§c§§d§a§e' THEN error := TRUE; END_IF;
LIST_INSERT(tmp, 9, 'f', L1);
IF L1 <> '§b§c§§d§a§e§§§f' THEN error := TRUE; END_IF;
LIST_INSERT(tmp, 0, '1', L1);
IF L1 <> '§1§b§c§§d§a§e§§§f' THEN error := TRUE; END_IF;
END_FUNCTION_BLOCK

(* POU X_TEST/test_list_next, ST *)
FUNCTION_BLOCK test_list_next
VAR_INPUT
END_VAR
VAR_OUTPUT
	error: BOOL;
END_VAR
VAR
	lx : LIST_NEXT;
	L1: STRING(LIST_LENGTH);
	tmp: BYTE;
END_VAR
IF error THEN RETURN; END_IF;
L1 := '§1§§3';
tmp := CODE('§',1);
lx(SEP := tmp, LIST := L1);
IF lx.LEL <> '1' THEN error := TRUE; END_IF;
IF lx.NUL = TRUE THEN error := TRUE; END_IF;
lx(SEP := tmp, LIST := L1);
IF lx.LEL <> '' THEN error := TRUE; END_IF;
IF lx.NUL = TRUE THEN error := TRUE; END_IF;
lx(SEP := tmp, LIST := L1);
IF lx.LEL <> '3' THEN error := TRUE; END_IF;
IF lx.NUL = TRUE THEN error := TRUE; END_IF;
lx(SEP := tmp, LIST := L1);
IF lx.LEL <> '' THEN error := TRUE; END_IF;
IF lx.NUL = FALSE THEN error := TRUE; END_IF;
L1 := '§§';
lx(SEP := tmp, rst := TRUE, LIST := L1);
lx.rst := FALSE;
IF lx.LEL <> '' THEN error := TRUE; END_IF;
IF lx.NUL = TRUE THEN error := TRUE; END_IF;
lx(SEP := tmp,  LIST := L1);
IF lx.LEL <> '' THEN error := TRUE; END_IF;
IF lx.NUL = TRUE THEN error := TRUE; END_IF;
lx(SEP := tmp,  LIST := L1);
IF lx.LEL <> '' THEN error := TRUE; END_IF;
IF lx.NUL = FALSE THEN error := TRUE; END_IF;
L1 := '';
lx(SEP := tmp, rst := TRUE, LIST := L1);
lx.rst := FALSE;
IF lx.LEL <> '' THEN error := TRUE; END_IF;
IF lx.NUL = FALSE THEN error := TRUE; END_IF;
END_FUNCTION_BLOCK

(* POU X_TEST/test_list_retrieve, ST *)
FUNCTION_BLOCK test_list_retrieve
VAR_INPUT
END_VAR
VAR_OUTPUT
	error: BOOL;
END_VAR
VAR
	L1: STRING(LIST_LENGTH);
	tmp : BYTE;
END_VAR
IF error THEN RETURN; END_IF;
L1 := '§1§§3§4§5';
tmp := CODE('§',1);

IF LIST_RETRIEVE(tmp,0,L1) <> '' THEN error := TRUE; END_IF;
IF L1 <> '§1§§3§4§5' THEN error := TRUE; END_IF;
IF LIST_RETRIEVE(tmp,6,L1) <> '' THEN error := TRUE; END_IF;
IF L1 <> '§1§§3§4§5' THEN error := TRUE; END_IF;
IF LIST_RETRIEVE(tmp,1,L1) <> '1' THEN error := TRUE; END_IF;
IF L1 <> '§§3§4§5' THEN error := TRUE; END_IF;
IF LIST_RETRIEVE(tmp,4,L1) <> '5' THEN error := TRUE; END_IF;
IF L1 <> '§§3§4' THEN error := TRUE; END_IF;
IF LIST_RETRIEVE(tmp,1,L1) <> '' THEN error := TRUE; END_IF;
IF L1 <> '§3§4' THEN error := TRUE; END_IF;
L1 := '§§';
IF LIST_RETRIEVE(tmp,2,L1) <> '' THEN error := TRUE; END_IF;
IF L1 <> '§' THEN error := TRUE; END_IF;
IF LIST_RETRIEVE(tmp,2,L1) <> '' THEN error := TRUE; END_IF;
IF L1 <> '§' THEN error := TRUE; END_IF;
IF LIST_RETRIEVE(tmp,1,L1) <> '' THEN error := TRUE; END_IF;
IF L1 <> '' THEN error := TRUE; END_IF;
IF LIST_RETRIEVE(tmp,1,L1) <> '' THEN error := TRUE; END_IF;
END_FUNCTION_BLOCK

(* POU X_TEST/test_list_retrieve_last, ST *)
FUNCTION_BLOCK test_list_retrieve_last
VAR_INPUT
END_VAR
VAR_OUTPUT
	error: BOOL;
END_VAR
VAR
	L1: STRING(LIST_LENGTH);
	tmp : BYTE;
END_VAR
IF error THEN RETURN; END_IF;
L1 := '§1§§3§4§5§';
tmp := CODE('§',1);

IF LIST_RETRIEVE_LAST(tmp,L1) <> '' THEN error := TRUE; END_IF;
IF L1 <> '§1§§3§4§5' THEN error := TRUE; END_IF;
IF LIST_RETRIEVE_LAST(tmp,L1) <> '5' THEN error := TRUE; END_IF;
IF L1 <> '§1§§3§4' THEN error := TRUE; END_IF;
IF LIST_RETRIEVE_LAST(tmp,L1) <> '4' THEN error := TRUE; END_IF;
IF L1 <> '§1§§3' THEN error := TRUE; END_IF;
IF LIST_RETRIEVE_LAST(tmp,L1) <> '3' THEN error := TRUE; END_IF;
IF L1 <> '§1§' THEN error := TRUE; END_IF;
IF LIST_RETRIEVE_LAST(tmp,L1) <> '' THEN error := TRUE; END_IF;
IF L1 <> '§1' THEN error := TRUE; END_IF;
IF LIST_RETRIEVE_LAST(tmp,L1) <> '1' THEN error := TRUE; END_IF;
IF L1 <> '' THEN error := TRUE; END_IF;
IF LIST_RETRIEVE_LAST(tmp,L1) <> '' THEN error := TRUE; END_IF;
IF L1 <> '' THEN error := TRUE; END_IF;
END_FUNCTION_BLOCK

(* POU X_TEST/test_mid3, ST *)
FUNCTION_BLOCK test_mid3
VAR_INPUT
END_VAR
VAR_OUTPUT
	error : BOOL;
END_VAR
VAR
END_VAR
IF MID3(0,0,0) <> 0 THEN error := TRUE; END_IF;
IF MID3(0,0,1) <> 0 THEN error := TRUE; END_IF;
IF MID3(1,0,0) <> 0 THEN error := TRUE; END_IF;
IF MID3(0,1,0) <> 0 THEN error := TRUE; END_IF;
IF MID3(1,1,0) <> 1 THEN error := TRUE; END_IF;
IF MID3(0,1,1) <> 1 THEN error := TRUE; END_IF;
IF MID3(1,0,1) <> 1 THEN error := TRUE; END_IF;
IF MID3(0,1,2) <> 1 THEN error := TRUE; END_IF;
IF MID3(0,2,1) <> 1 THEN error := TRUE; END_IF;
IF MID3(1,0,2) <> 1 THEN error := TRUE; END_IF;
IF MID3(1,2,0) <> 1 THEN error := TRUE; END_IF;
IF MID3(2,0,1) <> 1 THEN error := TRUE; END_IF;
IF MID3(2,1,0) <> 1 THEN error := TRUE; END_IF;
END_FUNCTION_BLOCK

(* POU X_TEST/test_set_date, ST *)
FUNCTION_BLOCK test_set_date
VAR_INPUT
END_VAR
VAR_OUTPUT
	error: BOOL;
END_VAR
VAR

END_VAR
IF SET_DATE(1970,1,1) <> d#1970-1-1 THEN error := TRUE; END_IF;
IF SET_DATE(1970,2,28) <> d#1970-2-28 THEN error := TRUE; END_IF;
IF SET_DATE(1970,3,1) <> d#1970-3-1 THEN error := TRUE; END_IF;
IF SET_DATE(1970,12,31) <> d#1970-12-31 THEN error := TRUE; END_IF;
IF SET_DATE(1971,1,1) <> d#1971-1-1 THEN error := TRUE; END_IF;
IF SET_DATE(1971,2,28) <> d#1971-2-28 THEN error := TRUE; END_IF;
IF SET_DATE(1971,3,1) <> d#1971-3-1 THEN error := TRUE; END_IF;
IF SET_DATE(1971,12,31) <> d#1971-12-31 THEN error := TRUE; END_IF;
IF SET_DATE(1972,1,1) <> d#1972-1-1 THEN error := TRUE; END_IF;
IF SET_DATE(1972,2,28) <> d#1972-2-28 THEN error := TRUE; END_IF;
IF SET_DATE(1972,2,29) <> d#1972-2-29 THEN error := TRUE; END_IF;
IF SET_DATE(1972,3,1) <> d#1972-3-1 THEN error := TRUE; END_IF;
IF SET_DATE(1972,12,31) <> d#1972-12-31 THEN error := TRUE; END_IF;
IF SET_DATE(1973,1,1) <> d#1973-1-1 THEN error := TRUE; END_IF;
IF SET_DATE(1973,2,28) <> d#1973-2-28 THEN error := TRUE; END_IF;
IF SET_DATE(1973,3,1) <> d#1973-3-1 THEN error := TRUE; END_IF;
IF SET_DATE(1973,12,31) <> d#1973-12-31 THEN error := TRUE; END_IF;
IF SET_DATE(1999,12,31) <> d#1999-12-31 THEN error := TRUE; END_IF;
IF SET_DATE(2000,1,1) <> d#2000-1-1 THEN error := TRUE; END_IF;
IF SET_DATE(2000,1,31) <> d#2000-1-31 THEN error := TRUE; END_IF;
IF SET_DATE(2000,2,1) <> d#2000-2-1 THEN error := TRUE; END_IF;
IF SET_DATE(2000,2,29) <> d#2000-2-29 THEN error := TRUE; END_IF;
IF SET_DATE(2000,3,1) <> d#2000-3-1 THEN error := TRUE; END_IF;
IF SET_DATE(2000,3,31) <> d#2000-3-31 THEN error := TRUE; END_IF;
IF SET_DATE(2000,4,1) <> d#2000-4-1 THEN error := TRUE; END_IF;
IF SET_DATE(2000,4,30) <> d#2000-4-30 THEN error := TRUE; END_IF;
IF SET_DATE(2000,5,1) <> d#2000-5-1 THEN error := TRUE; END_IF;
IF SET_DATE(2000,5,31) <> d#2000-5-31 THEN error := TRUE; END_IF;
IF SET_DATE(2000,6,1) <> d#2000-6-1 THEN error := TRUE; END_IF;
IF SET_DATE(2000,6,30) <> d#2000-6-30 THEN error := TRUE; END_IF;
IF SET_DATE(2000,7,1) <> d#2000-7-1 THEN error := TRUE; END_IF;
IF SET_DATE(2000,7,31) <> d#2000-7-31 THEN error := TRUE; END_IF;
IF SET_DATE(2000,8,1) <> d#2000-8-1 THEN error := TRUE; END_IF;
IF SET_DATE(2000,8,31) <> d#2000-8-31 THEN error := TRUE; END_IF;
IF SET_DATE(2000,9,1) <> d#2000-9-1 THEN error := TRUE; END_IF;
IF SET_DATE(2000,9,30) <> d#2000-9-30 THEN error := TRUE; END_IF;
IF SET_DATE(2000,10,1) <> d#2000-10-1 THEN error := TRUE; END_IF;
IF SET_DATE(2000,10,31) <> d#2000-10-31 THEN error := TRUE; END_IF;
IF SET_DATE(2000,11,1) <> d#2000-11-1 THEN error := TRUE; END_IF;
IF SET_DATE(2000,11,30) <> d#2000-11-30 THEN error := TRUE; END_IF;
IF SET_DATE(2000,12,1) <> d#2000-12-1 THEN error := TRUE; END_IF;
IF SET_DATE(2000,12,31) <> d#2000-12-31 THEN error := TRUE; END_IF;
IF SET_DATE(2099,12,31) <> d#2099-12-31 THEN error := TRUE; END_IF;
END_FUNCTION_BLOCK

(* POU String/TICKER, ST *)
FUNCTION_BLOCK TICKER

VAR_INPUT
	N : INT;
	PT : TIME;
END_VAR

VAR_IN_OUT
	Text : STRING(STRING_LENGTH);
END_VAR

VAR_OUTPUT
	Display : STRING(STRING_LENGTH);
END_VAR
VAR
	delay : TP;
	step : INT;
END_VAR

(*
version 1.2	29. mar. 2008
programmer 	hugo
tested by		tobias

Ticker sends a substring of text with length N every TD Milliseconds to generate a ticker. 

*)
(* generate next ticker when delay is low *)
IF N < LEN(text) THEN
	IF NOT delay.Q THEN
		(* increase step for next tick *)
		step := step + 1;
		IF step > LEN(text) THEN step := 1; END_IF;
		(* extract dispay from text *)
		display := MID(text, N, step);
		(* set delay timer for next tick *)
		delay(in := TRUE, PT := PT);
	ELSE;
		(* execute delay timer *)
		delay(in := FALSE);
	END_IF;
ELSE
	display := text;
END_IF;
(* revision history
hm	4. dec. 2007	rev 1.0
	original version

hm	15. dec. 2007	rev 1.1
	step now starts at 1 instaed of 0

hm	29. mar. 2008	rev 1.2
	changed STRING to STRING(STRING_LENGTH)
*)
END_FUNCTION_BLOCK

(* POU Time&Date/TIMECHECK, ST *)
FUNCTION TIMECHECK : BOOL
VAR_INPUT
	TD : TOD;
	START : TOD;
	STOP : TOD;
END_VAR


(*
version 1.0	19. jul. 2009
programmer 	oscat
tested by		oscat

this function retruns true if the daytime TD is between start and stop and returns true if so.
if you want to generate an event to span over midnight, start timemust be later than the stop time.

*)
IF stop < start THEN
	TIMECHECK := start <= TD OR TD < stop;
ELSE
	TIMECHECK := start <= TD AND TD < stop;
END_IF;



(* revision history
hm 19. jul. 2009	rev 1.0
	original release

*)
END_FUNCTION

(* POU Logic/FF edge triggered/TOGGLE, ST *)
FUNCTION_BLOCK TOGGLE
VAR_INPUT
	CLK : BOOL;
	rst : BOOL;
END_VAR
VAR_OUTPUT
	Q : BOOL;
END_VAR
VAR
	edge : BOOL;
END_VAR

(*
version 1.1	30. oct. 2008
programmer 	hugo
tested by	oscat

toggle flip flop the output changes state with every rising edge of clk.

*)
IF rst THEN
	q := 0;
ELSIF clk AND NOT edge THEN
	Q := NOT Q;
END_IF;
edge := clk;

(* revision history

hm	13.9.2007		rev 1.0
	original version

hm	30. oct. 2008	rev 1.1
	deleted unnecessary init

*)
END_FUNCTION_BLOCK

(* POU Logic/generators/TONOF, ST *)
FUNCTION_BLOCK TONOF
VAR_INPUT
	IN : BOOL;
	  T_ON,T_OFF : TIME;
END_VAR
VAR_OUTPUT
	Q : BOOL;
END_VAR
VAR
   X : TON;
   old: BOOL;
   mode: BOOL;
END_VAR

(*
version 1.2	21. jul 2009
programmer 	hugo
tested by		tobias

TONOF generated a TON and TOF Delay for the Input N TON (T1) and TOF (T2) can be configured separately
*)
IF IN XOR old THEN
  X(IN := FALSE, PT := SEL(IN,T_OFF,T_ON));
  mode := IN;
  old := IN;
END_IF;
X(IN := TRUE);
IF X.Q THEN Q := mode;END_IF;

(* revision history
hm	10. dec 2007	rev 1.0
	original version

hm	17. sep. 2007	rev 1.1
	improved performance

hm	21. jul. 2009	rev 1.2
	fixed a timing probelm


*)
END_FUNCTION_BLOCK

(* POU Engineering/signal processing/TREND, ST *)
FUNCTION_BLOCK TREND
VAR_INPUT
	X : REAL;
END_VAR
VAR_OUTPUT
	Q : BOOL;
	TU : BOOL;
	TD : BOOL;
	D : REAL;
END_VAR
VAR
	last_X: REAL;
END_VAR

(*
version 1.0	21. aug. 2009
programmer 	hugo
tested by		oscat

trend analyses the trend of a input signal.
The Output Q is True if the input X is >= last_X and is false if the input X is <= last_X
in addition to the trend the output TU will be high for one cycle to signal a rising of the input value X
and  TD will signal a decreasing value on the input X.
in case of a change the output D will show the delta of the input to the last input value.

*)
TU := X > last_X;
TD := X < last_X;
Q := TU OR TD;
D := X - LAST_X;

last_X := X;



(* revision history
hm	21. aug. 2009	rev 1.0
	original version

*)
END_FUNCTION_BLOCK

(* POU Mathematical/Geometry/TRIANGLE_A, ST *)
FUNCTION TRIANGLE_A : REAL
VAR_INPUT
	S1 : REAL;
	A : REAL;
	S2 : REAL;
	S3 : REAL;
END_VAR


(*
version 1.2	10. mar. 2009
programmer 	hugo
tested by		tobias

triangle_A calculates the Area of a triangle.
if any input is 0 it will be neglected and the are will be calculated from eiter:
two sides and an angle (s1 and S2 and the angle A1) or 3 sides.


*)
IF A = 0.0 THEN
	TRIANGLE_A := SQRT((s1+s2+S3) * (s1+s2-S3) * (S2+S3-S1) * (S3+S1-S2)) * 0.25;
ELSE
	TRIANGLE_A := S1 * S2 * SIN(RAD(A)) * 0.5;
END_IF;

(* revision histroy
hm	16. oct 2007	rev 1.0
	original version

hm	22. feb 2008	rev 1.1
	improved performance

hm	10. mar. 2009	rev 1.2
	changed syntax of real constants to 0.0

*)
END_FUNCTION

(* POU String/TRIM1, ST *)
FUNCTION TRIM1 : STRING(STRING_LENGTH)
VAR_INPUT
	str : STRING(STRING_LENGTH);
END_VAR
VAR
	pos: INT;
END_VAR

(*
version 1.2	29. mar. 2008
programmer 	hugo
tested by		tobias

the function replaces all multiple blanks within a string by only one blank.
leading and ending blanks will be deleted

*)
TRIM1 := str;
REPEAT
	pos := FIND(trim1,'  ');
	IF pos > 0 THEN TRIM1 := REPLACE(TRIM1,' ',2,pos); END_IF;
UNTIL pos = 0	END_REPEAT;
(* beginning and ending blanks need to be stripped off *)
IF LEFT(trim1,1) = ' ' THEN trim1 := DELETE(trim1,1,1); END_IF;
IF RIGHT(trim1,1) = ' ' THEN trim1 := DELETE(trim1,1,LEN(trim1)); END_IF;


(* revision histroy
hm	4. feb. 2008    rev 1.0
	original release

hm	20. mar. 2008	rev 1.1
	avoid to call replace with pos = 0 because some systems will produce an error

hm	29. mar. 2008	rev 1.2
	changed STRING to STRING(STRING_LENGTH)
*)
END_FUNCTION

(* POU String/TRIME, ST *)
FUNCTION TRIME : STRING(string_length)
VAR_INPUT
	str : STRING(STRING_LENGTH);
END_VAR


(*
version 1.0	28. mar. 2008
programmer 	hugo
tested by	tobias

this function deletes all leading and ending blanks of a string.

*)
TRIME := str;
(* beginning blanks need to be stripped off *)
WHILE LEFT(TRIME,1) = ' ' DO
	TRIME := DELETE(TRIME,1,1);
END_WHILE;

(* ending blanks need to be stripped off *)
WHILE RIGHT(TRIME,1) = ' ' DO
	TRIME := DELETE(TRIME,1,LEN(TRIME));
END_WHILE;


(* revision histroy
hm	28. mar. 2008	rev 1.0
	original release

*)
END_FUNCTION

(* POU Engineering/automation/TUNE, ST *)
FUNCTION_BLOCK TUNE
VAR_INPUT
	SET : BOOL;
	SU, SD : BOOL;
	RST : BOOL;
END_VAR
VAR_INPUT CONSTANT
	SS : REAL := 0.1;
	Limit_L : REAL;
	LIMIT_H : REAL := 100.0;
	RST_val : REAL;
	SET_val : REAL := 100.0;
	T1 : TIME := T#500ms;
	T2 : TIME := T#2s;
	S1 : REAL := 2.0;
	S2 : REAL := 10.0;
END_VAR
VAR_OUTPUT
	Y : REAL;
END_VAR
VAR
	tx : DWORD;
	start, start2 : DWORD;
	state : INT;
	in : BOOL;
	step : REAL;
	SPEED : REAL;
	Y_start : REAL;
	Y_start2: REAL;
END_VAR

(*
version 1.2	11. mar. 2009
programmer 	hugo
tested by		tobias

tune generates an output signal which is set by input switches.
up to 4 switsches can be used to tune the signal up or down.

*)
(* read system time *)
tx := T_PLC_MS();

IF rst THEN
	Y := RST_val;
	state := 0;
ELSIF set THEN
	Y := SET_val;
	state := 0;
ELSIF state > 0 THEN
	(* key has been pushed state machine operating *)
	(* first read the correct input *)
	IF state = 1 THEN
		(* step up *)
		in := su;
	ELSE
		(* step down *)
		in := sd;
	END_IF;
	(* check for single step operation *)
	IF NOT in AND tx - start <= TIME_TO_DWORD(T1) THEN
		Y := Y_start + step;
		state := 0;
	(* check if fast ramp needs to be generated *)
	ELSIF in AND tx - start >= TIME_TO_DWORD(T2) THEN
		Y := Y_start2 + DWORD_TO_REAL(tx - start2) * s2 / speed;
	(* check if slow ramp needs to be generated *)
	ELSIF in AND tx - start >= TIME_TO_DWORD(T1) THEN
		Y := Y_start + DWORD_TO_REAL(tx - start - TIME_TO_DWORD(T1)) * S1 / speed;
		start2 := tx;
		Y_start2 := Y;
	ELSIF NOT in THEN
		state := 0;
	END_IF;
ELSIF su THEN
	(* slow step up *)
	state := 1;
	start := tx;
	step := ss;
	speed := 1000.0;
	Y_start := Y;
ELSIF sd THEN
	(* slow step down *)
	state := 2;
	start := tx;
	step := -ss;
	speed := -1000.0;
	Y_start := Y;
END_IF;

(* make sure output does not exceed limits *)
Y := LIMIT(LIMIT_L, Y, LIMIT_H);

(* revision history
hm	3.11.2007		rev 1.0
	original version

hm	16. mar. 2008	rev 1.1
	added type conversions to avoid warnings under codesys 3.0

hm	11. mar. 2009	rev 1.2
	real constants updated to new systax using dot																																																																																																																																																																																																																																																																																																																																																																																																																																																																																																																																																																																																																																																																																																																																																																																																																																																																																																																																																																																																																																																											

*)
END_FUNCTION_BLOCK

(* POU Engineering/automation/TUNE2, ST *)
FUNCTION_BLOCK TUNE2
VAR_INPUT
	SET : BOOL;
	SU, SD : BOOL;
	FU, FD : BOOL;
	RST : BOOL;
END_VAR
VAR_INPUT CONSTANT
	SS : REAL := 0.1;
	FS : REAL := 5.0;
	Limit_L : REAL;
	LIMIT_H : REAL := 100.0;
	RST_val : REAL;
	SET_val : REAL := 100.0;
	TR : TIME := T#500ms;
	S1 : REAL := 2.0;
	S2 : REAL := 10.0;
END_VAR
VAR_OUTPUT
	Y : REAL;
END_VAR
VAR
	tx : DWORD;
	start : DWORD;
	state : INT;
	in : BOOL;
	step : REAL;
	SPEED : REAL;
	Y_start : REAL;
END_VAR

(*
version 1.2	11. mar. 2009
programmer 	hugo
tested by		tobias

tune2 generates an output signal which is set by input switches.
up to 4 switsches can be used to tune the signal up or down.

*)
(* read system time *)
tx := T_PLC_MS();

IF rst THEN
	Y := RST_val;
	state := 0;
ELSIF set THEN
	Y := SET_val;
	state := 0;
ELSIF state > 0 THEN
	(* key has been pushed state machine operating *)
	(* first read the correct input *)
	CASE state OF
		1 :	(* slow up *)
			in := su;
		2 :	(* slow down *)
			in := sd;
		3 :	(* fast up *)
			in := fu;
		4 :	(* fast down *)
			in := fd;
	END_CASE;
	(* check for single step operation *)
	IF NOT in AND tx - start <= TIME_TO_DWORD(TR) THEN
		Y := Y_start + step;
		state := 0;
	(* check if ramp needs to be generated *)
	ELSIF in AND tx - start >= TIME_TO_DWORD(TR) THEN
		Y := Y_start + DWORD_TO_REAL(tx - start - TIME_TO_DWORD(TR)) * speed;
	ELSIF NOT in THEN
		state := 0;
	END_IF;
ELSIF su THEN
	(* slow step up *)
	state := 1;
	start := tx;
	step := ss;
	speed := s1 * 1.0E-3;
	Y_start := Y;
ELSIF sd THEN
	(* slow step down *)
	state := 2;
	start := tx;
	step := -ss;
	speed := -s1 * 1.0E-3;
	Y_start := Y;
ELSIF fu THEN
	(* fast step up *)
	state := 3;
	start := tx;
	step := fs;
	speed := s2 * 1.0E-3;
	y_start := Y;
ELSIF fd THEN
	(* fast step down *)
	state := 4;
	start := tx;
	step := -fs;
	speed := -s2 * 1.0E-3;
	y_start := Y;
END_IF;

(* make sure output does not exceed limits *)
Y := LIMIT(LIMIT_L, Y, LIMIT_H);

(* revision history
hm	3.11.2007		rev 1.0
	original version

hm	16. 3. 2008	rev 1.1
	added type conversions to avoid warnings in codesys 3.0
	improved performance

hm	11. mar. 2009	rev 1.2
	real constants updated to new systax using dot																																																																																																																																																																																																																																																																																																																																																																																																																																																																																																																																																																																																																																																																																																																																																																																																																																																																																																																																																																																																																																																											

*)
END_FUNCTION_BLOCK

(* POU Mathematical/Vektormathematik/V3_ABS, ST *)
FUNCTION V3_ABS : REAL
VAR_INPUT
	A : Vector_3;
END_VAR


(*
version 1.0	11 dec 2007
programmer 	hugo
tested by		tobias

this function calculates the length of a vectors in a 3 dimensional space

*)
V3_ABS := SQRT(A.X * A.X + A.Y * A.Y + A.Z * A.Z);


(* revision history
hm		11 dec 2007	rev 1.0
	original version

*)
END_FUNCTION

(* POU Mathematical/Vektormathematik/V3_ADD, ST *)
FUNCTION V3_ADD : vector_3
VAR_INPUT
	A : Vector_3;
	B : Vector_3;
END_VAR


(*
version 1.0	11 dec 2007
programmer 	hugo
tested by		tobias

this function adds two vectors in a 3 dimensional space

*)
V3_ADD.X := A.X + B.X;
V3_ADD.Y := A.Y + B.Y;
V3_ADD.Z := A.Z + B.Z;



(* revision history
hm		11 dec 2007	rev 1.0
	original version

*)
END_FUNCTION

(* POU Mathematical/Vektormathematik/V3_ANG, ST *)
FUNCTION V3_ANG : REAL
VAR_INPUT
	A : Vector_3;
	B : Vector_3;
END_VAR
VAR
	d : REAL;
END_VAR

(*
version 1.1	10. mar. 2009
programmer 	hugo
tested by		tobias

this function calculates the angle between two vectors in a 3 dimensional space

*)
d := V3_ABS(A) * V3_ABS(B);
IF d > 0 THEN
	V3_ANG := ACOS(LIMIT(-1.0, V3_DPRO(A, B) / d,1.0));
END_IF;

(* revision history
hm	11. dec. 2007	rev 1.0
	original version

hm	10. mar. 2009	rev 1.1
	changed syntax of real constants to 0.0

*)
END_FUNCTION

(* POU Mathematical/Vektormathematik/V3_DPRO, ST *)
FUNCTION V3_DPRO : REAL
VAR_INPUT
	A : Vector_3;
	B : Vector_3;
END_VAR


(*
version 1.0	11 dec 2007
programmer 	hugo
tested by		tobias

this function calculates the dot product of two vectors in 3 dimensional space

*)
V3_DPRO := A.X * B.X + A.Y * B.Y + A.Z * B.Z;


(* revision history
hm		11 dec 2007	rev 1.0
	original version

*)
END_FUNCTION

(* POU Mathematical/Vektormathematik/V3_NORM, ST *)
FUNCTION V3_NORM : vector_3
VAR_INPUT
	A : Vector_3;
END_VAR
VAR
	la: REAL;
END_VAR

(*
version 1.1	10. mar. 2009
programmer 	hugo
tested by		tobias

this function generates a vectors with absolute length 1 from a vector A in a 3 dimensional space

*)
la := V3_ABS(A);
IF la > 0.0 THEN
	V3_NORM := V3_SMUL(A, 1.0 / la);
END_IF;

(* revision history
hm	11 dec 2007	rev 1.0
	original version

hm	10. mar. 2009	rev 1.1
	changed syntax of real constants to 0.0

*)
END_FUNCTION

(* POU Mathematical/Vektormathematik/V3_SMUL, ST *)
FUNCTION V3_SMUL : vector_3
VAR_INPUT
	A : Vector_3;
	M : REAL;
END_VAR


(*
version 1.0	11 dec 2007
programmer 	hugo
tested by		tobias

this function multiplies a vectors in a 3 dimensional space with a skalar M

*)
V3_SMUL.X := A.X * M;
V3_SMUL.Y := A.Y * M;
V3_SMUL.Z := A.Z * M;



(* revision history
hm		11 dec 2007	rev 1.0
	original version

*)
END_FUNCTION

(* POU Mathematical/Vektormathematik/V3_NUL, ST *)
FUNCTION V3_NUL : BOOL
VAR_INPUT
	A : Vector_3;
END_VAR


(*
version 1.1	10. mar. 2009
programmer 	hugo
tested by		tobias

this function checks if a vectors in a null Vector

*)
V3_NUL := A.X = 0.0 AND A.Y = 0.0 AND A.Z = 0.0;



(* revision history
hm	12 dec 2007	rev 1.0
	original version

hm	10. mar. 2009	rev 1.1
	changed syntax of real constants to 0.0

*)
END_FUNCTION

(* POU Mathematical/Vektormathematik/V3_PAR, ST *)
FUNCTION V3_PAR : BOOL
VAR_INPUT
	A : Vector_3;
	B : Vector_3;
END_VAR


(*
version 1.1	10. mar. 2009
programmer 	hugo
tested by		tobias

this function checks if two vectors in a 3 dimensional space are parallel.
which means the two vectors have the same direction

*)
V3_PAR := V3_ABS(V3_XPRO(A, B)) = 0.0;



(* revision history
hm	11 dec 2007	rev 1.0
	original version

hm	10. mar. 2009	rev 1.1
	changed syntax of real constants to 0.0

*)
END_FUNCTION

(* POU Mathematical/Vektormathematik/V3_XPRO, ST *)
FUNCTION V3_XPRO : vector_3
VAR_INPUT
	A : Vector_3;
	B : Vector_3;
END_VAR


(*
version 1.0	11 dec 2007
programmer 	hugo
tested by		tobias

this function adds two vectors in a 3 dimensional space

*)
V3_XPRO.X := A.Y * B.Z - A.Z * B.Y;
V3_XPRO.Y := A.Z * B.X - A.X * B.Z;
V3_XPRO.Z := A.X * B.Y - A.Y * B.X;



(* revision history
hm		11 dec 2007	rev 1.0
	original version

*)
END_FUNCTION

(* POU Mathematical/Vektormathematik/V3_REV, ST *)
FUNCTION V3_REV : vector_3
VAR_INPUT
	A : Vector_3;
END_VAR


(*
version 1.0	11 dec 2007
programmer 	hugo
tested by		tobias

this function reverses a vector in a 3 dimensional space

*)
V3_REV.X := -A.X;
V3_REV.Y := -A.Y;
V3_REV.Z := -A.Z;



(* revision history
hm		11 dec 2007	rev 1.0
	original version

*)
END_FUNCTION

(* POU Mathematical/Vektormathematik/V3_SUB, ST *)
FUNCTION V3_SUB : vector_3
VAR_INPUT
	A : Vector_3;
	B : Vector_3;
END_VAR


(*
version 1.0	11 dec 2007
programmer 	hugo
tested by		tobias

this function subtracts two vectors in a 3 dimensional space
V3_SUB = A - B

*)
V3_SUB.X := A.X - B.X;
V3_SUB.Y := A.Y - B.Y;
V3_SUB.Z := A.Z - B.Z;



(* revision history
hm		11 dec 2007	rev 1.0
	original version

*)
END_FUNCTION

(* POU Mathematical/Vektormathematik/V3_XANG, ST *)
FUNCTION V3_XANG : REAL
VAR_INPUT
	A : Vector_3;
END_VAR
VAR
	la: REAL;
END_VAR

(*
version 1.1	10. mar. 2009
programmer 	hugo
tested by		tobias

this function calculates the angle between the X-axis and a vectors in a 3 dimensional space

*)
la := V3_ABS(a);
IF la > 0.0 THEN
	V3_XANG := ACOS(A.X / la);
END_IF;

(* revision history
hm	11 dec 2007	rev 1.0
	original version

hm	10. mar. 2009	rev 1.1
	changed syntax of real constants to 0.0

*)
END_FUNCTION

(* POU Mathematical/Vektormathematik/V3_YANG, ST *)
FUNCTION V3_YANG : REAL
VAR_INPUT
	A : Vector_3;
END_VAR
VAR
	la: REAL;
END_VAR

(*
version 1.1	10. mar. 2009
programmer 	hugo
tested by		tobias

this function calculates the angle between the Y-axis and a vectors in a 3 dimensional space

*)
la := V3_ABS(a);
IF la > 0.0 THEN
	V3_YANG := ACOS(A.Y / la);
END_IF;

(* revision history
hm	11 dec 2007	rev 1.0
	original version

hm	10. mar. 2009	rev 1.1
	changed syntax of real constants to 0.0

*)
END_FUNCTION

(* POU Mathematical/Vektormathematik/V3_ZANG, ST *)
FUNCTION V3_ZANG : REAL
VAR_INPUT
	A : Vector_3;
END_VAR
VAR
	la: REAL;
END_VAR

(*
version 1.1	10. mar. 2009
programmer 	hugo
tested by		tobias

this function calculates the angle between the Z-axis and a vectors in a 3 dimensional space

*)
la := V3_ABS(a);
IF la > 0.0 THEN
	V3_ZANG := ACOS(A.Z / la);
END_IF;

(* revision history
hm	11 dec 2007	rev 1.0
	original version

hm	10. mar. 2009	rev 1.1
	changed syntax of real constants to 0.0

*)
END_FUNCTION

(* POU Mathematical/WINDOW, ST *)
FUNCTION WINDOW : BOOL
VAR_INPUT
	low : REAL;
	in : REAL;
	high : REAL;
END_VAR


(*
	version 1.1	22 jan 2007
	programmer 	hugo
	tested BY	tobias

this checks a signal if the signal is between the upper and lower limit
*)
WINDOW := in < high AND in > low;


(* revision history
hm	22.1.2007	rev 1.1
	changed the order of inputs to low, in, high

*)
END_FUNCTION

(* POU Mathematical/WINDOW2, ST *)
FUNCTION WINDOW2 : BOOL
VAR_INPUT
	LOW : REAL;
	IN : REAL;
	HIGH : REAL;
END_VAR


(*
	version 1.0	31 oct 2007
	programmer 	hugo
	tested BY	tobias

this checks a signal if the signal is between the upper and lower limit including the two limits
*)
WINDOW2 := IN >= LOW AND IN <= HIGH;


(* revision history
hm	31.10.2007	rev 1.0
	original version

*)
END_FUNCTION

(* POU Logic/gate logic/WORD_OF_BYTE, ST *)
FUNCTION WORD_OF_BYTE : WORD
VAR_INPUT
	B1 : BYTE;
	B0 : BYTE;
END_VAR


(*
version 1.4	18. jul. 2009
programmer 	hugo
tested by		tobias

this function creates a word from 2 individual bytes

*)
WORD_OF_BYTE := SHL(BYTE_TO_WORD(B1),8) OR BYTE_TO_WORD(B0);

(* revision history
hm	24. jan 2007	rev 1.0
	original version

hm	2. jan 2008	rev 1.1
	improved performance

hm	19. feb 2008	rev 1.2
	replaced and with or for better compatibility

hm	23. apr. 2008	rev 1.3
	reverse order of inputs to be more logical

hm	18. jul. 2009	rev 1.4
	added type conversions for compatibility reasons

*)
END_FUNCTION

(* POU Logic/gate logic/WORD_OF_DWORD, ST *)
FUNCTION WORD_OF_DWORD : WORD
VAR_INPUT
	in : DWORD;
	N : BYTE;
END_VAR


(*
version 1.2	30. oct. 2008
programmer 	hugo
tested by	oscat

this function extracts a single word from the nth position from right (right is lowest byte)
the lower word (starting with Bit0 from in) is selected with N=0.
*)
WORD_OF_DWORD := DWORD_TO_WORD(SHR(in,SHL(n,4)));

(* revision history
hm	17. jan 2007	rev 1.0
	original version

hm	2. jan 2008		rev 1.1
	improved performance

hm	30. oct. 2008	rev 1.2
	improved performance
*)
END_FUNCTION

(* POU Engineering/signal processing/WORD_TO_RANGE, ST *)
FUNCTION WORD_TO_RANGE : REAL
VAR_INPUT
	X : WORD;
	low : REAL;
	high : REAL;
END_VAR


(*
version 1.1	10. mar. 2009
programmer 	hugo
tested by		tobias

Word_to_Range converts a Byte into a real between low and high.

*)
WORD_TO_RANGE := (high - low) * WORD_TO_REAL(X) * 0.00001525902189669640 + low;


(* revision history
hm	9. jan 2008	rev 1.0
	original version

hm	10. mar. 2009	rev 1.1
	improved code
*)
END_FUNCTION
